FUNCTION F_TimeStToFileStr : STRING
VAR_INPUT
	timeToConvert:TIMESTRUCT;
END_VAR
VAR
	s1:STRING;
END_VAR
//Converts a timestruct variable to a string that can be used as file name

s1:=WORD_TO_STRING(timeToConvert.wYear);
s1:=CONCAT(s1,WORD_TO_STRING(timeToConvert.wMonth));
s1:=CONCAT(s1,WORD_TO_STRING(timeToConvert.wDay));
s1:=CONCAT(s1,'_');
s1:=CONCAT(s1,WORD_TO_STRING(timeToConvert.wHour));
s1:=CONCAT(s1,'_');
s1:=CONCAT(s1,WORD_TO_STRING(timeToConvert.wMinute));
s1:=CONCAT(s1,'_');
s1:=CONCAT(s1,WORD_TO_STRING(timeToConvert.wSecond));

F_TimeStToFileStr:=s1;

END_FUNCTION

(* stored: Version 1.1.0.1, ProductVersion 3.1.4024.12
   POU F_TimeStToFileStr: Id {99713a09-b995-4949-be67-c869804266f1}, SpecialFunc None *)
